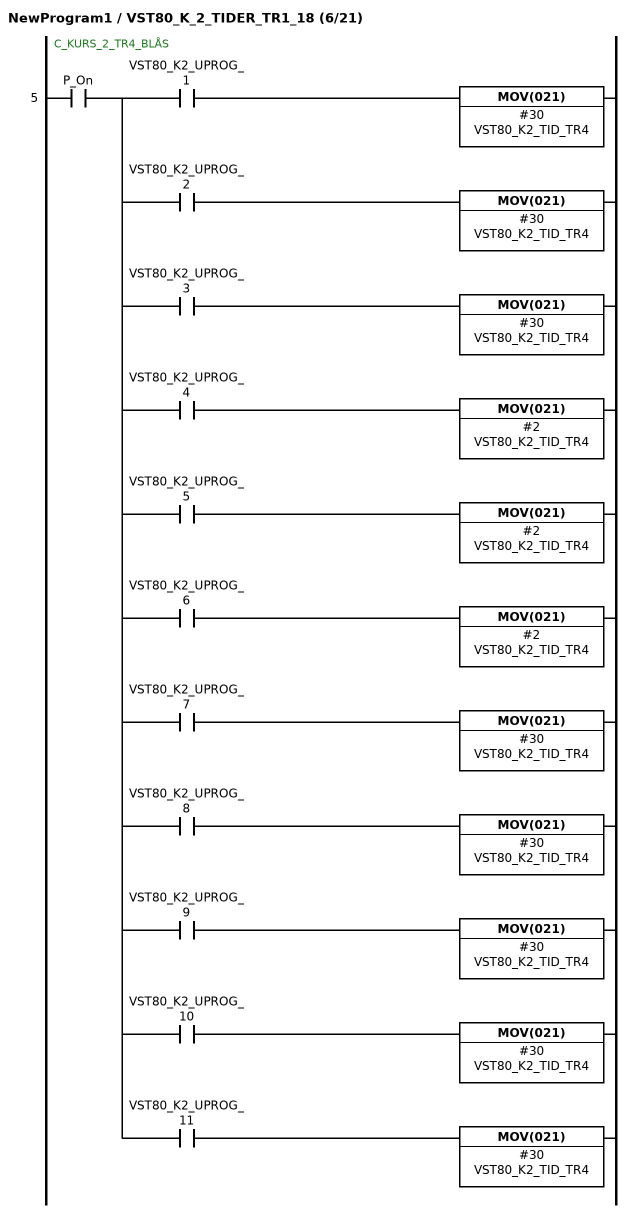
; [picture p168: NewProgram1 / VST80_K_2_TIDER_TR1_18, rungs 5-5]
; rung 5: C_KURS_2_TR4_BLÅS
LD P_On
OUT TR0
AND VST80_K2_UPROG_1
MOV(021) #30 VST80_K2_TID_TR4
LD TR0
AND VST80_K2_UPROG_2
MOV(021) #30 VST80_K2_TID_TR4
LD TR0
AND VST80_K2_UPROG_3
MOV(021) #30 VST80_K2_TID_TR4
LD TR0
AND VST80_K2_UPROG_4
MOV(021) #2 VST80_K2_TID_TR4
LD TR0
AND VST80_K2_UPROG_5
MOV(021) #2 VST80_K2_TID_TR4
LD TR0
AND VST80_K2_UPROG_6
MOV(021) #2 VST80_K2_TID_TR4
LD TR0
AND VST80_K2_UPROG_7
MOV(021) #30 VST80_K2_TID_TR4
LD TR0
AND VST80_K2_UPROG_8
MOV(021) #30 VST80_K2_TID_TR4
LD TR0
AND VST80_K2_UPROG_9
MOV(021) #30 VST80_K2_TID_TR4
LD TR0
AND VST80_K2_UPROG_10
MOV(021) #30 VST80_K2_TID_TR4
LD TR0
AND VST80_K2_UPROG_11
MOV(021) #30 VST80_K2_TID_TR4

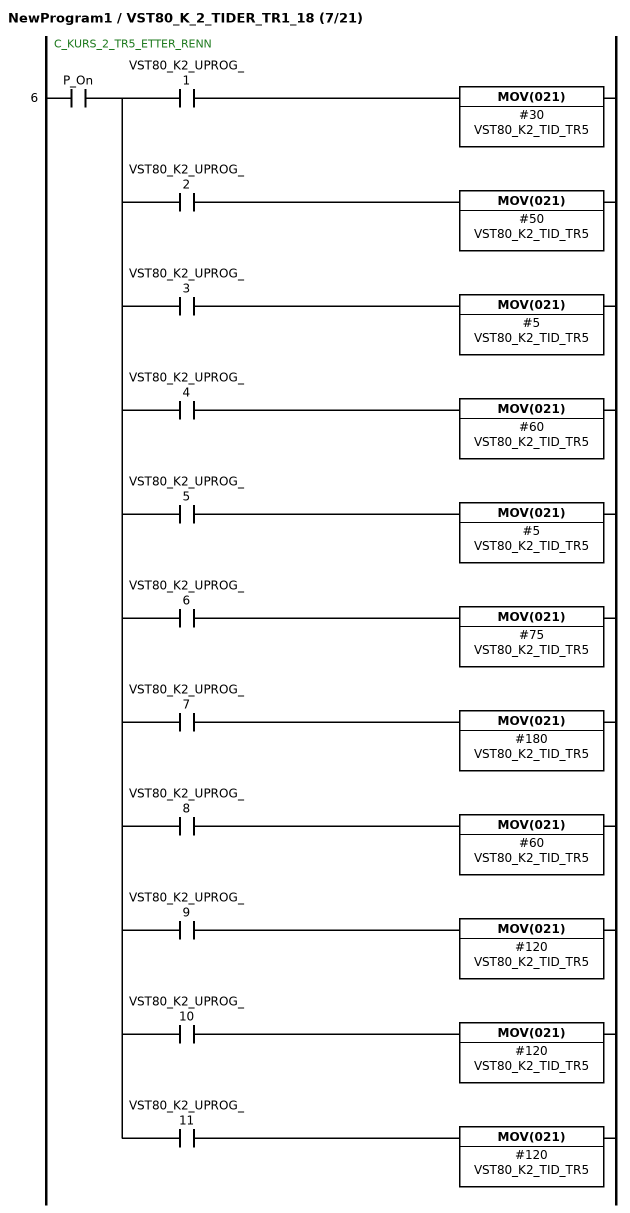
; rung 6: C_KURS_2_TR5_ETTER_RENN
LD P_On
OUT TR0
AND VST80_K2_UPROG_1
MOV(021) #30 VST80_K2_TID_TR5
LD TR0
AND VST80_K2_UPROG_2
MOV(021) #50 VST80_K2_TID_TR5
LD TR0
AND VST80_K2_UPROG_3
MOV(021) #5 VST80_K2_TID_TR5
LD TR0
AND VST80_K2_UPROG_4
MOV(021) #60 VST80_K2_TID_TR5
LD TR0
AND VST80_K2_UPROG_5
MOV(021) #5 VST80_K2_TID_TR5
LD TR0
AND VST80_K2_UPROG_6
MOV(021) #75 VST80_K2_TID_TR5
LD TR0
AND VST80_K2_UPROG_7
MOV(021) #180 VST80_K2_TID_TR5
LD TR0
AND VST80_K2_UPROG_8
MOV(021) #60 VST80_K2_TID_TR5
LD TR0
AND VST80_K2_UPROG_9
MOV(021) #120 VST80_K2_TID_TR5
LD TR0
AND VST80_K2_UPROG_10
MOV(021) #120 VST80_K2_TID_TR5
LD TR0
AND VST80_K2_UPROG_11
MOV(021) #120 VST80_K2_TID_TR5

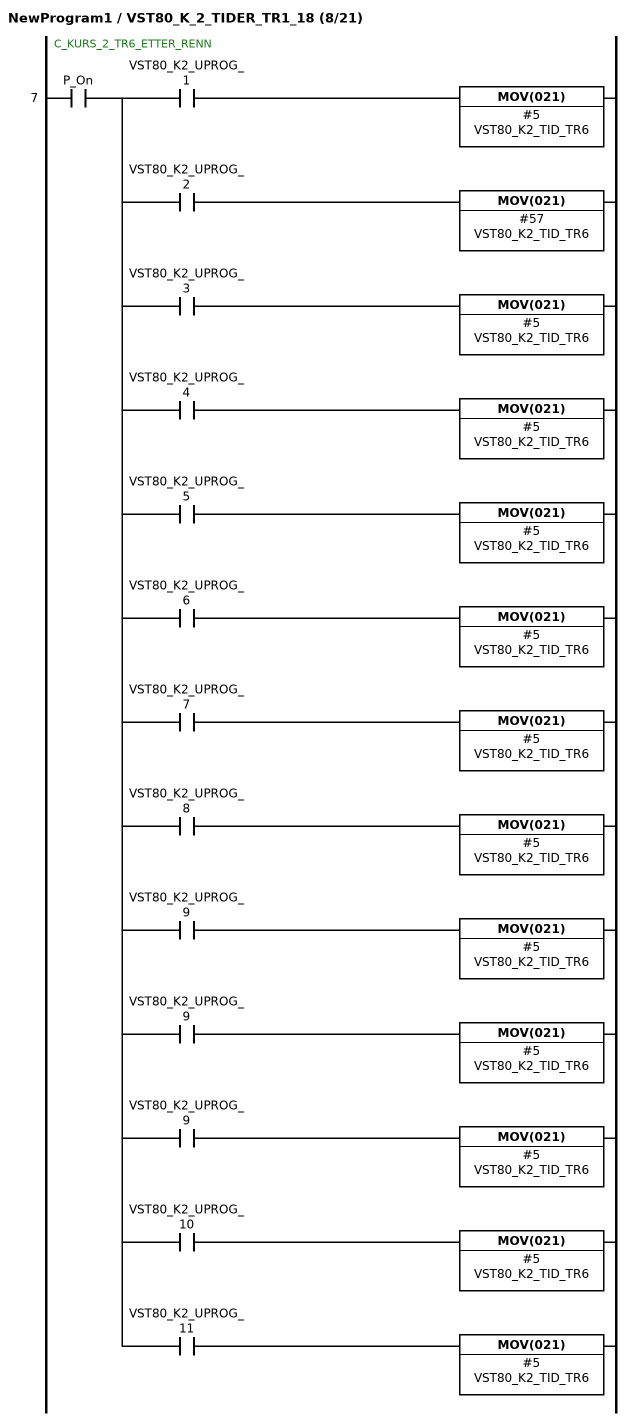
; rung 7: C_KURS_2_TR6_ETTER_RENN
LD P_On
OUT TR0
AND VST80_K2_UPROG_1
MOV(021) #5 VST80_K2_TID_TR6
LD TR0
AND VST80_K2_UPROG_2
MOV(021) #57 VST80_K2_TID_TR6
LD TR0
AND VST80_K2_UPROG_3
MOV(021) #5 VST80_K2_TID_TR6
LD TR0
AND VST80_K2_UPROG_4
MOV(021) #5 VST80_K2_TID_TR6
LD TR0
AND VST80_K2_UPROG_5
MOV(021) #5 VST80_K2_TID_TR6
LD TR0
AND VST80_K2_UPROG_6
MOV(021) #5 VST80_K2_TID_TR6
LD TR0
AND VST80_K2_UPROG_7
MOV(021) #5 VST80_K2_TID_TR6
LD TR0
AND VST80_K2_UPROG_8
MOV(021) #5 VST80_K2_TID_TR6
LD TR0
AND VST80_K2_UPROG_9
MOV(021) #5 VST80_K2_TID_TR6
LD TR0
AND VST80_K2_UPROG_9
MOV(021) #5 VST80_K2_TID_TR6
LD TR0
AND VST80_K2_UPROG_9
MOV(021) #5 VST80_K2_TID_TR6
LD TR0
AND VST80_K2_UPROG_10
MOV(021) #5 VST80_K2_TID_TR6
LD TR0
AND VST80_K2_UPROG_11
MOV(021) #5 VST80_K2_TID_TR6

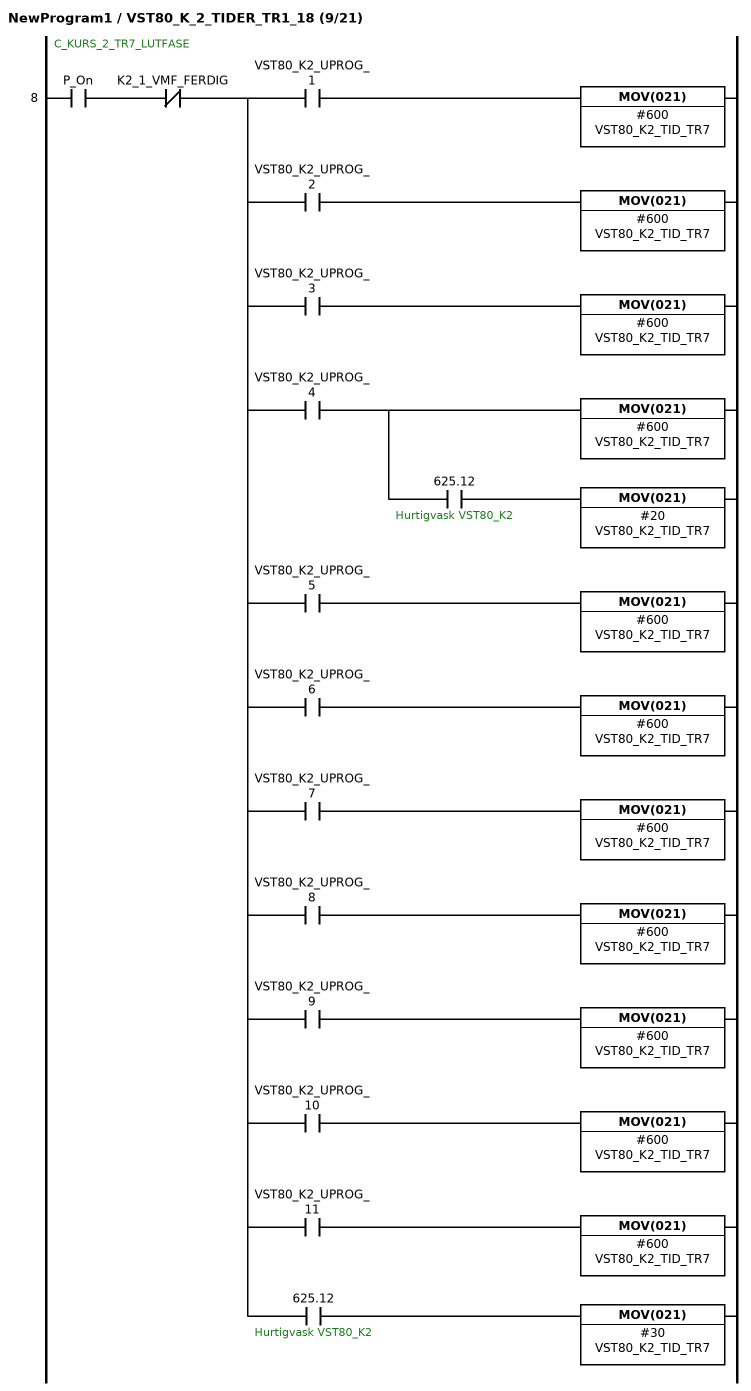
; rung 8: C_KURS_2_TR7_LUTFASE
LD P_On
ANDNOT K2_1_VMF_FERDIG
OUT TR0
AND VST80_K2_UPROG_1
MOV(021) #600 VST80_K2_TID_TR7
LD TR0
AND VST80_K2_UPROG_2
MOV(021) #600 VST80_K2_TID_TR7
LD TR0
AND VST80_K2_UPROG_3
MOV(021) #600 VST80_K2_TID_TR7
LD TR0
AND VST80_K2_UPROG_4
MOV(021) #600 VST80_K2_TID_TR7
AND 625.12  ; Hurtigvask VST80_K2
MOV(021) #20 VST80_K2_TID_TR7
LD TR0
AND VST80_K2_UPROG_5
MOV(021) #600 VST80_K2_TID_TR7
LD TR0
AND VST80_K2_UPROG_6
MOV(021) #600 VST80_K2_TID_TR7
LD TR0
AND VST80_K2_UPROG_7
MOV(021) #600 VST80_K2_TID_TR7
LD TR0
AND VST80_K2_UPROG_8
MOV(021) #600 VST80_K2_TID_TR7
LD TR0
AND VST80_K2_UPROG_9
MOV(021) #600 VST80_K2_TID_TR7
LD TR0
AND VST80_K2_UPROG_10
MOV(021) #600 VST80_K2_TID_TR7
LD TR0
AND VST80_K2_UPROG_11
MOV(021) #600 VST80_K2_TID_TR7
LD TR0
AND 625.12  ; Hurtigvask VST80_K2
MOV(021) #30 VST80_K2_TID_TR7

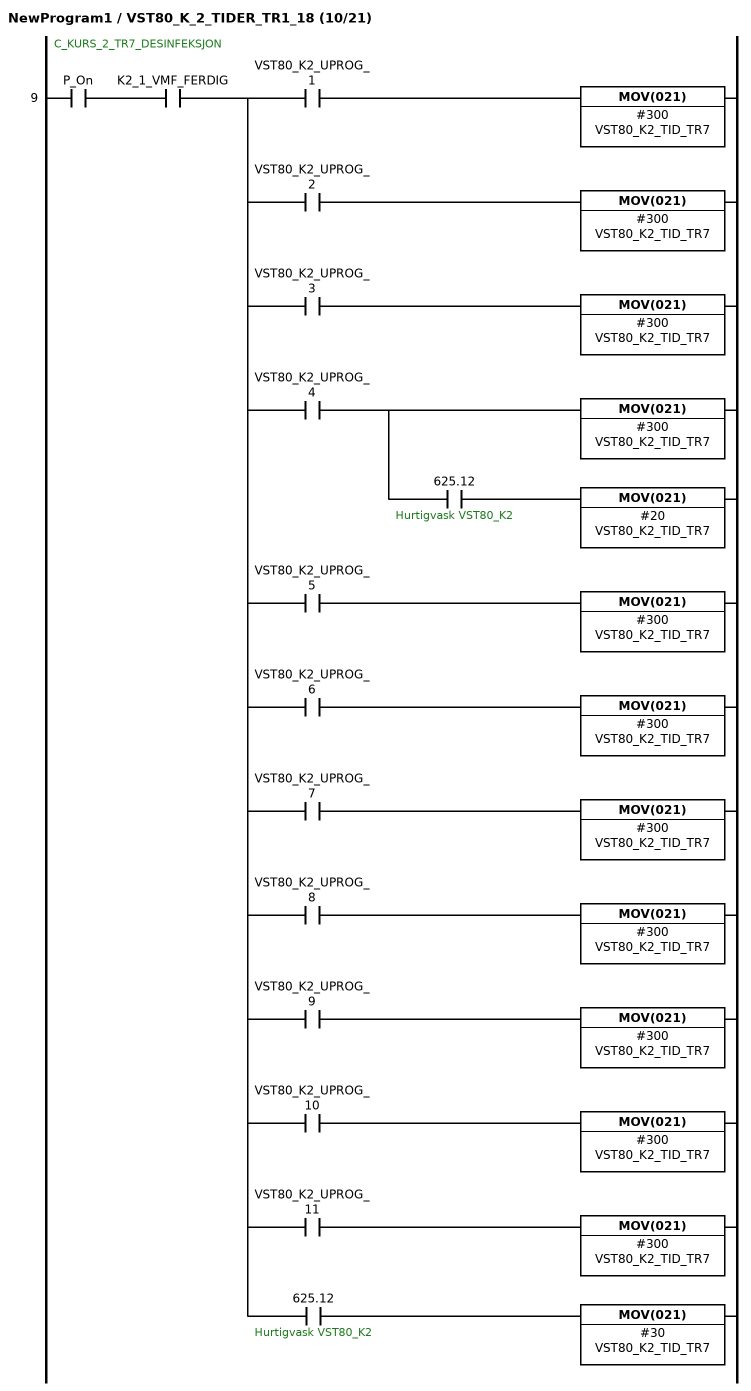
; rung 9: C_KURS_2_TR7_DESINFEKSJON
LD P_On
AND K2_1_VMF_FERDIG
OUT TR0
AND VST80_K2_UPROG_1
MOV(021) #300 VST80_K2_TID_TR7
LD TR0
AND VST80_K2_UPROG_2
MOV(021) #300 VST80_K2_TID_TR7
LD TR0
AND VST80_K2_UPROG_3
MOV(021) #300 VST80_K2_TID_TR7
LD TR0
AND VST80_K2_UPROG_4
MOV(021) #300 VST80_K2_TID_TR7
AND 625.12  ; Hurtigvask VST80_K2
MOV(021) #20 VST80_K2_TID_TR7
LD TR0
AND VST80_K2_UPROG_5
MOV(021) #300 VST80_K2_TID_TR7
LD TR0
AND VST80_K2_UPROG_6
MOV(021) #300 VST80_K2_TID_TR7
LD TR0
AND VST80_K2_UPROG_7
MOV(021) #300 VST80_K2_TID_TR7
LD TR0
AND VST80_K2_UPROG_8
MOV(021) #300 VST80_K2_TID_TR7
LD TR0
AND VST80_K2_UPROG_9
MOV(021) #300 VST80_K2_TID_TR7
LD TR0
AND VST80_K2_UPROG_10
MOV(021) #300 VST80_K2_TID_TR7
LD TR0
AND VST80_K2_UPROG_11
MOV(021) #300 VST80_K2_TID_TR7
LD TR0
AND 625.12  ; Hurtigvask VST80_K2
MOV(021) #30 VST80_K2_TID_TR7

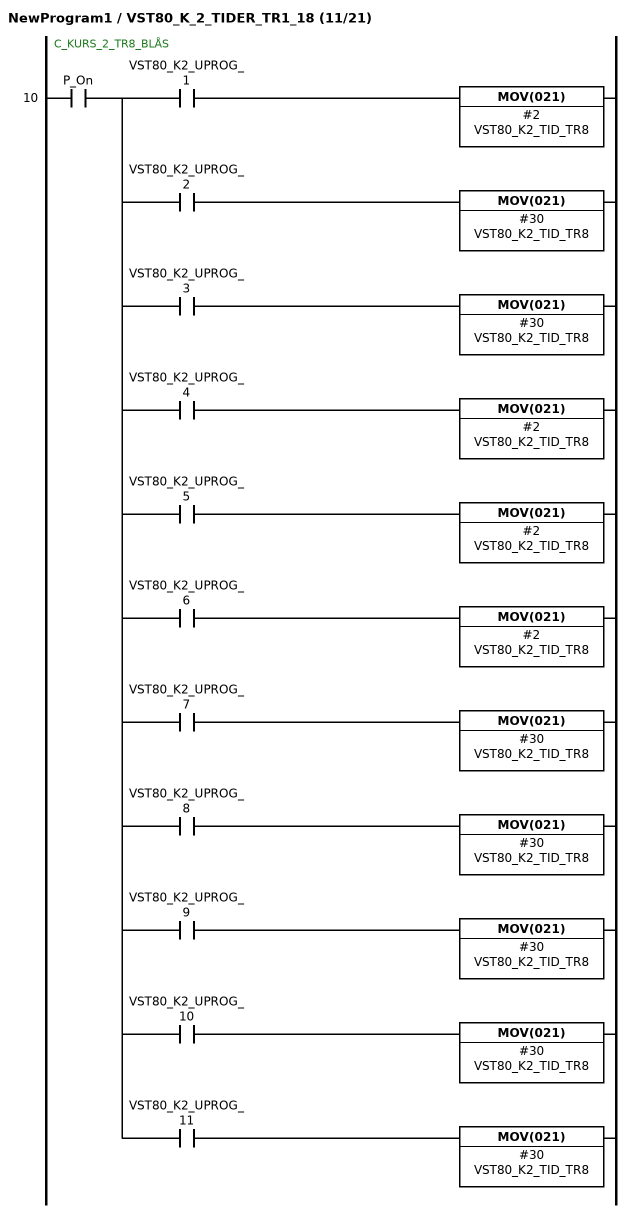
; rung 10: C_KURS_2_TR8_BLÅS
LD P_On
OUT TR0
AND VST80_K2_UPROG_1
MOV(021) #2 VST80_K2_TID_TR8
LD TR0
AND VST80_K2_UPROG_2
MOV(021) #30 VST80_K2_TID_TR8
LD TR0
AND VST80_K2_UPROG_3
MOV(021) #30 VST80_K2_TID_TR8
LD TR0
AND VST80_K2_UPROG_4
MOV(021) #2 VST80_K2_TID_TR8
LD TR0
AND VST80_K2_UPROG_5
MOV(021) #2 VST80_K2_TID_TR8
LD TR0
AND VST80_K2_UPROG_6
MOV(021) #2 VST80_K2_TID_TR8
LD TR0
AND VST80_K2_UPROG_7
MOV(021) #30 VST80_K2_TID_TR8
LD TR0
AND VST80_K2_UPROG_8
MOV(021) #30 VST80_K2_TID_TR8
LD TR0
AND VST80_K2_UPROG_9
MOV(021) #30 VST80_K2_TID_TR8
LD TR0
AND VST80_K2_UPROG_10
MOV(021) #30 VST80_K2_TID_TR8
LD TR0
AND VST80_K2_UPROG_11
MOV(021) #30 VST80_K2_TID_TR8

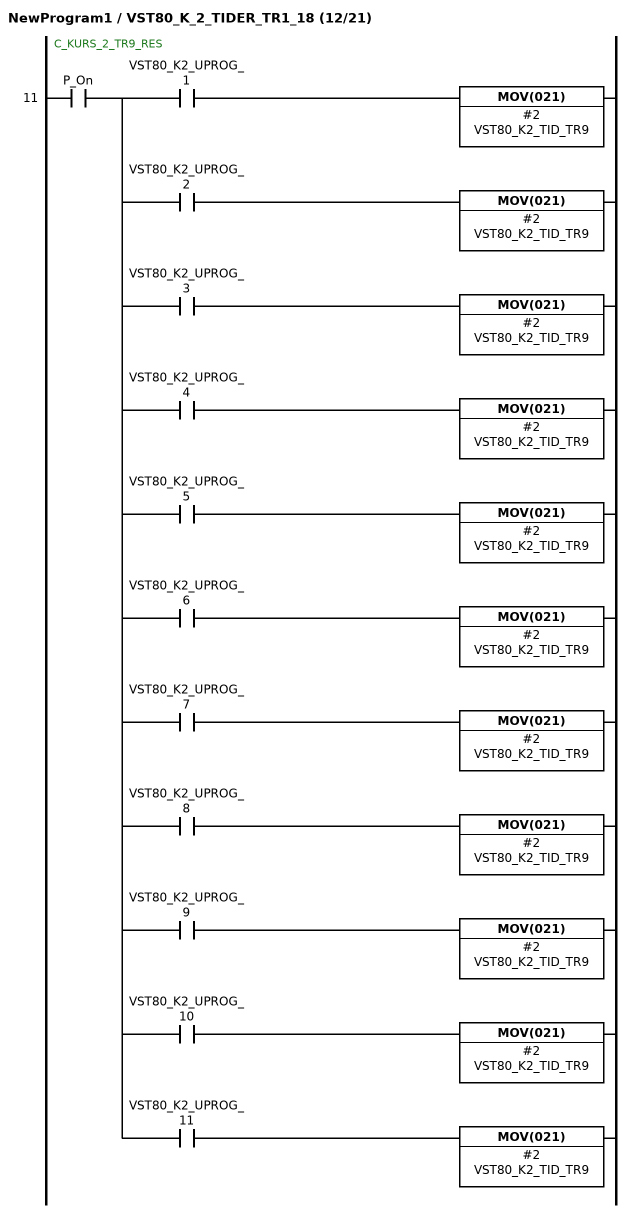
; rung 11: C_KURS_2_TR9_RES
LD P_On
OUT TR0
AND VST80_K2_UPROG_1
MOV(021) #2 VST80_K2_TID_TR9
LD TR0
AND VST80_K2_UPROG_2
MOV(021) #2 VST80_K2_TID_TR9
LD TR0
AND VST80_K2_UPROG_3
MOV(021) #2 VST80_K2_TID_TR9
LD TR0
AND VST80_K2_UPROG_4
MOV(021) #2 VST80_K2_TID_TR9
LD TR0
AND VST80_K2_UPROG_5
MOV(021) #2 VST80_K2_TID_TR9
LD TR0
AND VST80_K2_UPROG_6
MOV(021) #2 VST80_K2_TID_TR9
LD TR0
AND VST80_K2_UPROG_7
MOV(021) #2 VST80_K2_TID_TR9
LD TR0
AND VST80_K2_UPROG_8
MOV(021) #2 VST80_K2_TID_TR9
LD TR0
AND VST80_K2_UPROG_9
MOV(021) #2 VST80_K2_TID_TR9
LD TR0
AND VST80_K2_UPROG_10
MOV(021) #2 VST80_K2_TID_TR9
LD TR0
AND VST80_K2_UPROG_11
MOV(021) #2 VST80_K2_TID_TR9

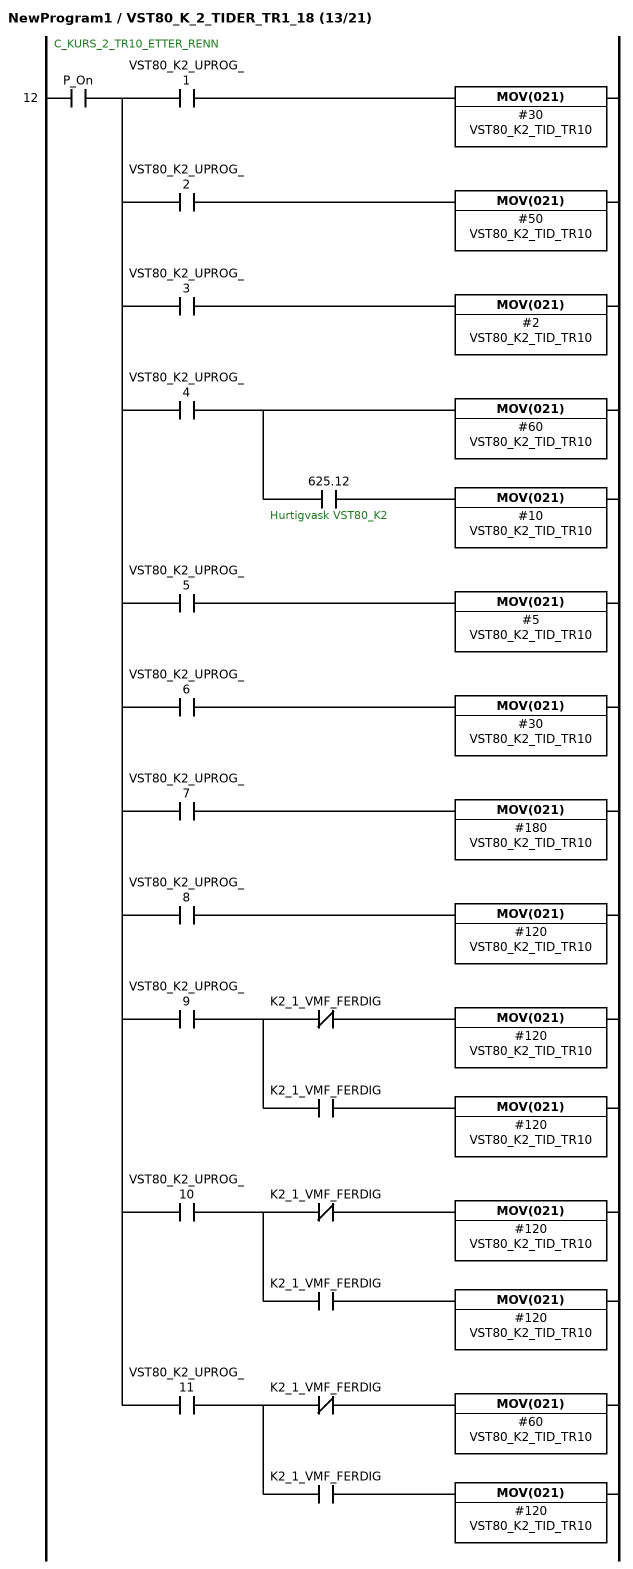
; rung 12: C_KURS_2_TR10_ETTER_RENN
LD P_On
OUT TR0
AND VST80_K2_UPROG_1
MOV(021) #30 VST80_K2_TID_TR10
LD TR0
AND VST80_K2_UPROG_2
MOV(021) #50 VST80_K2_TID_TR10
LD TR0
AND VST80_K2_UPROG_3
MOV(021) #2 VST80_K2_TID_TR10
LD TR0
AND VST80_K2_UPROG_4
MOV(021) #60 VST80_K2_TID_TR10
AND 625.12  ; Hurtigvask VST80_K2
MOV(021) #10 VST80_K2_TID_TR10
LD TR0
AND VST80_K2_UPROG_5
MOV(021) #5 VST80_K2_TID_TR10
LD TR0
AND VST80_K2_UPROG_6
MOV(021) #30 VST80_K2_TID_TR10
LD TR0
AND VST80_K2_UPROG_7
MOV(021) #180 VST80_K2_TID_TR10
LD TR0
AND VST80_K2_UPROG_8
MOV(021) #120 VST80_K2_TID_TR10
LD TR0
AND VST80_K2_UPROG_9
OUT TR1
ANDNOT K2_1_VMF_FERDIG
MOV(021) #120 VST80_K2_TID_TR10
LD TR1
AND K2_1_VMF_FERDIG
MOV(021) #120 VST80_K2_TID_TR10
LD TR0
AND VST80_K2_UPROG_10
OUT TR1
ANDNOT K2_1_VMF_FERDIG
MOV(021) #120 VST80_K2_TID_TR10
LD TR1
AND K2_1_VMF_FERDIG
MOV(021) #120 VST80_K2_TID_TR10
LD TR0
AND VST80_K2_UPROG_11
OUT TR0
ANDNOT K2_1_VMF_FERDIG
MOV(021) #60 VST80_K2_TID_TR10
LD TR0
AND K2_1_VMF_FERDIG
MOV(021) #120 VST80_K2_TID_TR10

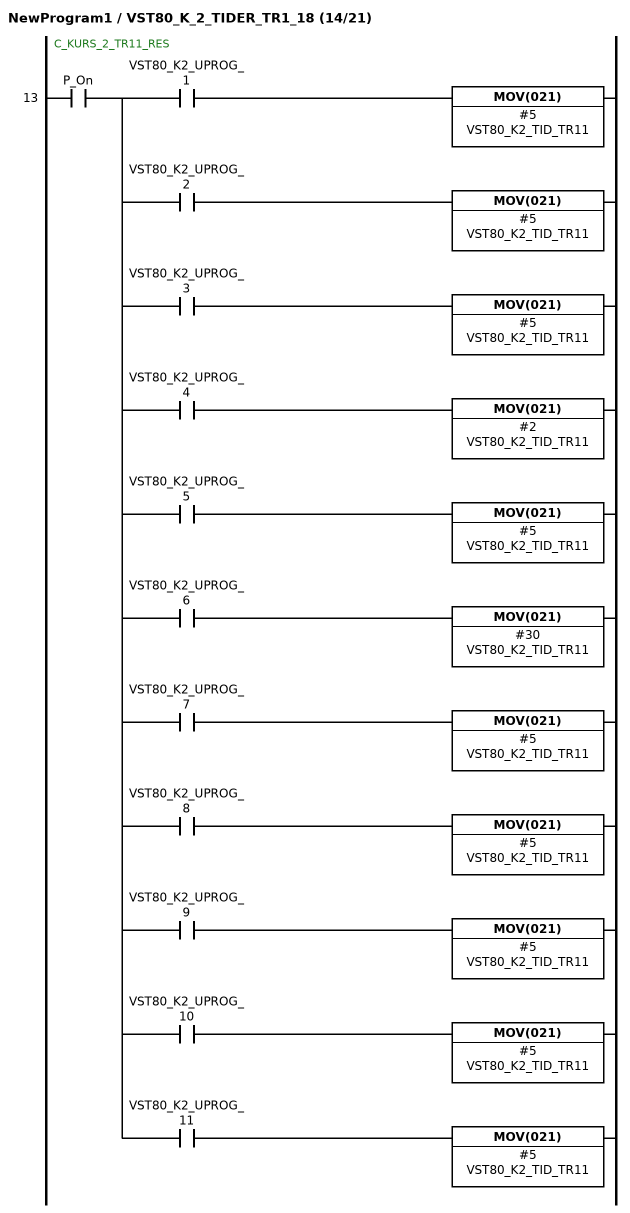
; rung 13: C_KURS_2_TR11_RES
LD P_On
OUT TR0
AND VST80_K2_UPROG_1
MOV(021) #5 VST80_K2_TID_TR11
LD TR0
AND VST80_K2_UPROG_2
MOV(021) #5 VST80_K2_TID_TR11
LD TR0
AND VST80_K2_UPROG_3
MOV(021) #5 VST80_K2_TID_TR11
LD TR0
AND VST80_K2_UPROG_4
MOV(021) #2 VST80_K2_TID_TR11
LD TR0
AND VST80_K2_UPROG_5
MOV(021) #5 VST80_K2_TID_TR11
LD TR0
AND VST80_K2_UPROG_6
MOV(021) #30 VST80_K2_TID_TR11
LD TR0
AND VST80_K2_UPROG_7
MOV(021) #5 VST80_K2_TID_TR11
LD TR0
AND VST80_K2_UPROG_8
MOV(021) #5 VST80_K2_TID_TR11
LD TR0
AND VST80_K2_UPROG_9
MOV(021) #5 VST80_K2_TID_TR11
LD TR0
AND VST80_K2_UPROG_10
MOV(021) #5 VST80_K2_TID_TR11
LD TR0
AND VST80_K2_UPROG_11
MOV(021) #5 VST80_K2_TID_TR11

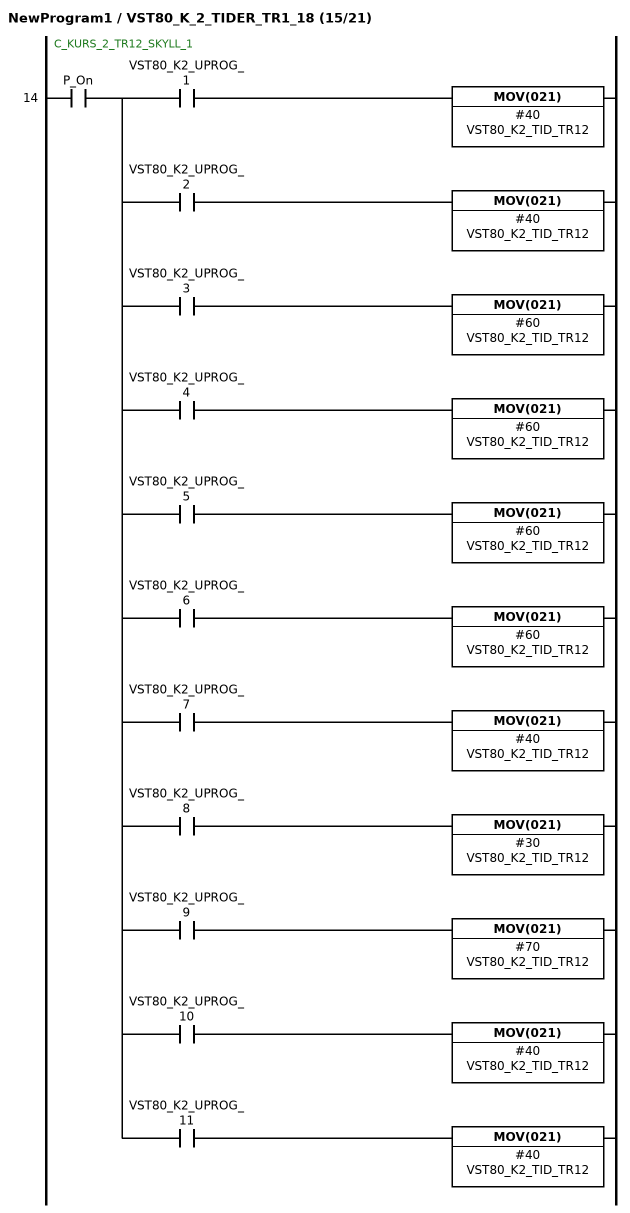
; rung 14: C_KURS_2_TR12_SKYLL_1
LD P_On
OUT TR0
AND VST80_K2_UPROG_1
MOV(021) #40 VST80_K2_TID_TR12
LD TR0
AND VST80_K2_UPROG_2
MOV(021) #40 VST80_K2_TID_TR12
LD TR0
AND VST80_K2_UPROG_3
MOV(021) #60 VST80_K2_TID_TR12
LD TR0
AND VST80_K2_UPROG_4
MOV(021) #60 VST80_K2_TID_TR12
LD TR0
AND VST80_K2_UPROG_5
MOV(021) #60 VST80_K2_TID_TR12
LD TR0
AND VST80_K2_UPROG_6
MOV(021) #60 VST80_K2_TID_TR12
LD TR0
AND VST80_K2_UPROG_7
MOV(021) #40 VST80_K2_TID_TR12
LD TR0
AND VST80_K2_UPROG_8
MOV(021) #30 VST80_K2_TID_TR12
LD TR0
AND VST80_K2_UPROG_9
MOV(021) #70 VST80_K2_TID_TR12
LD TR0
AND VST80_K2_UPROG_10
MOV(021) #40 VST80_K2_TID_TR12
LD TR0
AND VST80_K2_UPROG_11
MOV(021) #40 VST80_K2_TID_TR12

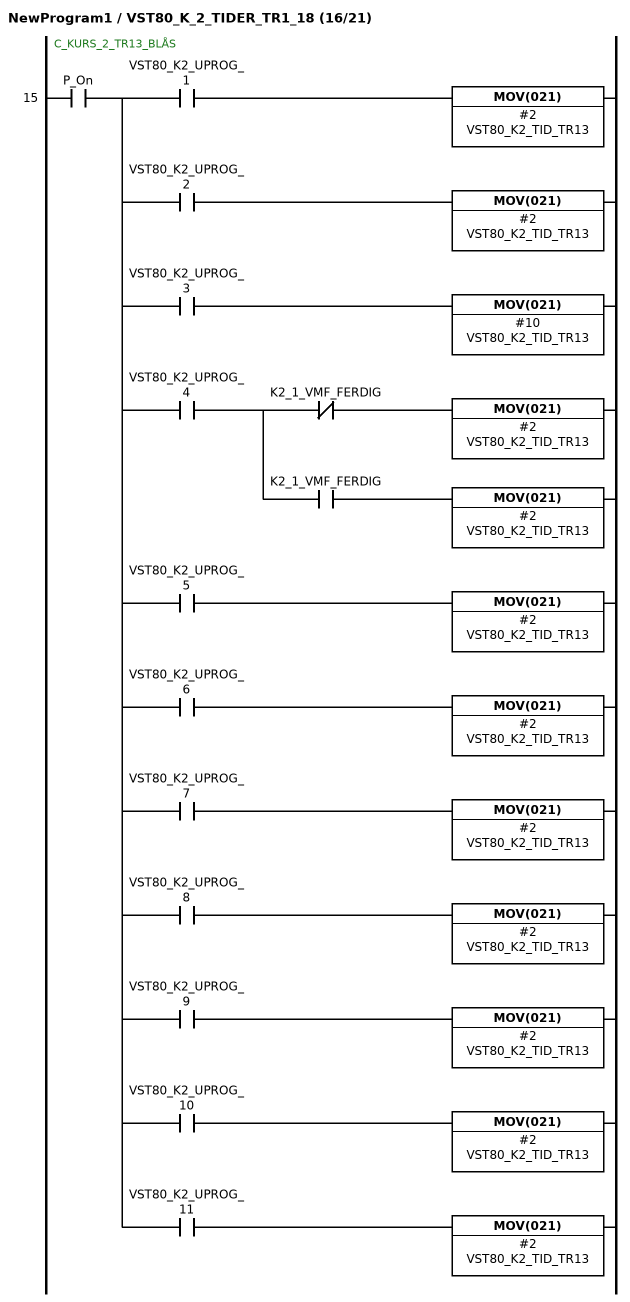
; rung 15: C_KURS_2_TR13_BLÅS
LD P_On
OUT TR0
AND VST80_K2_UPROG_1
MOV(021) #2 VST80_K2_TID_TR13
LD TR0
AND VST80_K2_UPROG_2
MOV(021) #2 VST80_K2_TID_TR13
LD TR0
AND VST80_K2_UPROG_3
MOV(021) #10 VST80_K2_TID_TR13
LD TR0
AND VST80_K2_UPROG_4
OUT TR1
ANDNOT K2_1_VMF_FERDIG
MOV(021) #2 VST80_K2_TID_TR13
LD TR1
AND K2_1_VMF_FERDIG
MOV(021) #2 VST80_K2_TID_TR13
LD TR0
AND VST80_K2_UPROG_5
MOV(021) #2 VST80_K2_TID_TR13
LD TR0
AND VST80_K2_UPROG_6
MOV(021) #2 VST80_K2_TID_TR13
LD TR0
AND VST80_K2_UPROG_7
MOV(021) #2 VST80_K2_TID_TR13
LD TR0
AND VST80_K2_UPROG_8
MOV(021) #2 VST80_K2_TID_TR13
LD TR0
AND VST80_K2_UPROG_9
MOV(021) #2 VST80_K2_TID_TR13
LD TR0
AND VST80_K2_UPROG_10
MOV(021) #2 VST80_K2_TID_TR13
LD TR0
AND VST80_K2_UPROG_11
MOV(021) #2 VST80_K2_TID_TR13

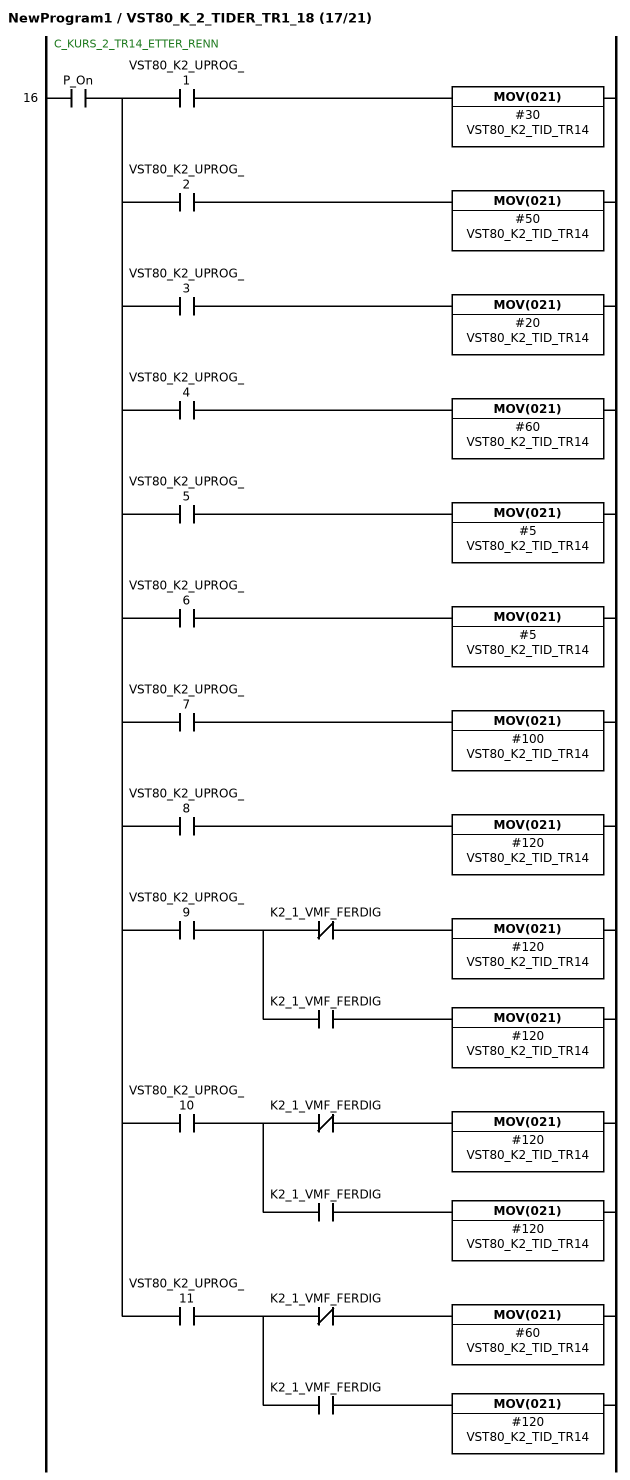
; rung 16: C_KURS_2_TR14_ETTER_RENN
LD P_On
OUT TR0
AND VST80_K2_UPROG_1
MOV(021) #30 VST80_K2_TID_TR14
LD TR0
AND VST80_K2_UPROG_2
MOV(021) #50 VST80_K2_TID_TR14
LD TR0
AND VST80_K2_UPROG_3
MOV(021) #20 VST80_K2_TID_TR14
LD TR0
AND VST80_K2_UPROG_4
MOV(021) #60 VST80_K2_TID_TR14
LD TR0
AND VST80_K2_UPROG_5
MOV(021) #5 VST80_K2_TID_TR14
LD TR0
AND VST80_K2_UPROG_6
MOV(021) #5 VST80_K2_TID_TR14
LD TR0
AND VST80_K2_UPROG_7
MOV(021) #100 VST80_K2_TID_TR14
LD TR0
AND VST80_K2_UPROG_8
MOV(021) #120 VST80_K2_TID_TR14
LD TR0
AND VST80_K2_UPROG_9
OUT TR1
ANDNOT K2_1_VMF_FERDIG
MOV(021) #120 VST80_K2_TID_TR14
LD TR1
AND K2_1_VMF_FERDIG
MOV(021) #120 VST80_K2_TID_TR14
LD TR0
AND VST80_K2_UPROG_10
OUT TR1
ANDNOT K2_1_VMF_FERDIG
MOV(021) #120 VST80_K2_TID_TR14
LD TR1
AND K2_1_VMF_FERDIG
MOV(021) #120 VST80_K2_TID_TR14
LD TR0
AND VST80_K2_UPROG_11
OUT TR0
ANDNOT K2_1_VMF_FERDIG
MOV(021) #60 VST80_K2_TID_TR14
LD TR0
AND K2_1_VMF_FERDIG
MOV(021) #120 VST80_K2_TID_TR14

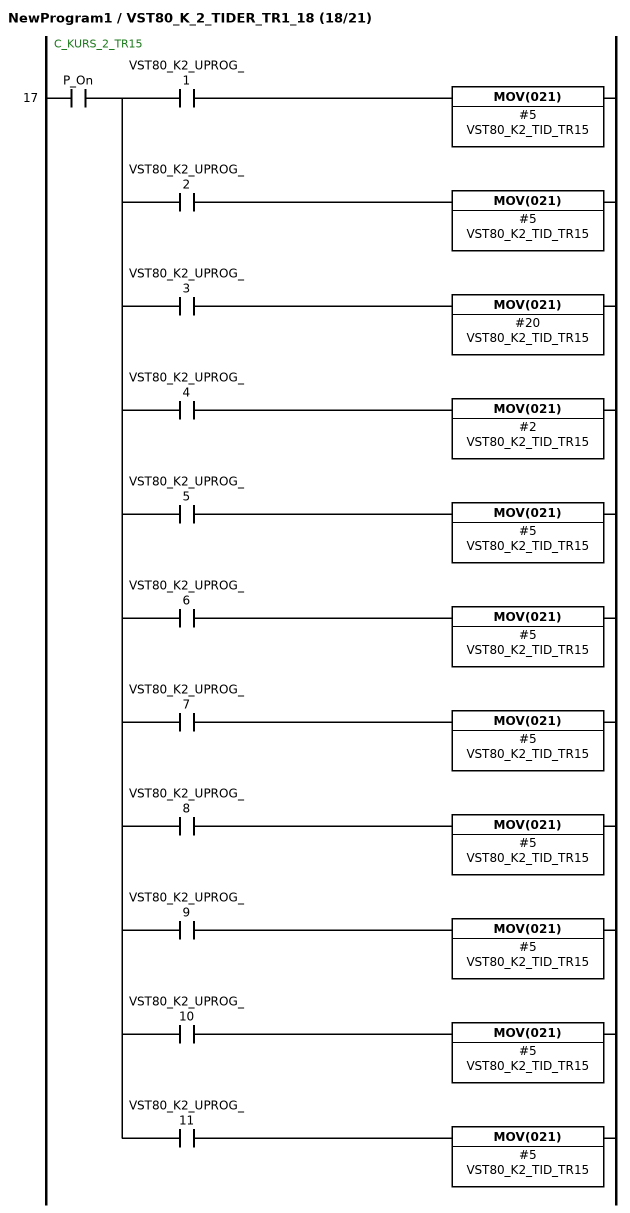
; rung 17: C_KURS_2_TR15
LD P_On
OUT TR0
AND VST80_K2_UPROG_1
MOV(021) #5 VST80_K2_TID_TR15
LD TR0
AND VST80_K2_UPROG_2
MOV(021) #5 VST80_K2_TID_TR15
LD TR0
AND VST80_K2_UPROG_3
MOV(021) #20 VST80_K2_TID_TR15
LD TR0
AND VST80_K2_UPROG_4
MOV(021) #2 VST80_K2_TID_TR15
LD TR0
AND VST80_K2_UPROG_5
MOV(021) #5 VST80_K2_TID_TR15
LD TR0
AND VST80_K2_UPROG_6
MOV(021) #5 VST80_K2_TID_TR15
LD TR0
AND VST80_K2_UPROG_7
MOV(021) #5 VST80_K2_TID_TR15
LD TR0
AND VST80_K2_UPROG_8
MOV(021) #5 VST80_K2_TID_TR15
LD TR0
AND VST80_K2_UPROG_9
MOV(021) #5 VST80_K2_TID_TR15
LD TR0
AND VST80_K2_UPROG_10
MOV(021) #5 VST80_K2_TID_TR15
LD TR0
AND VST80_K2_UPROG_11
MOV(021) #5 VST80_K2_TID_TR15

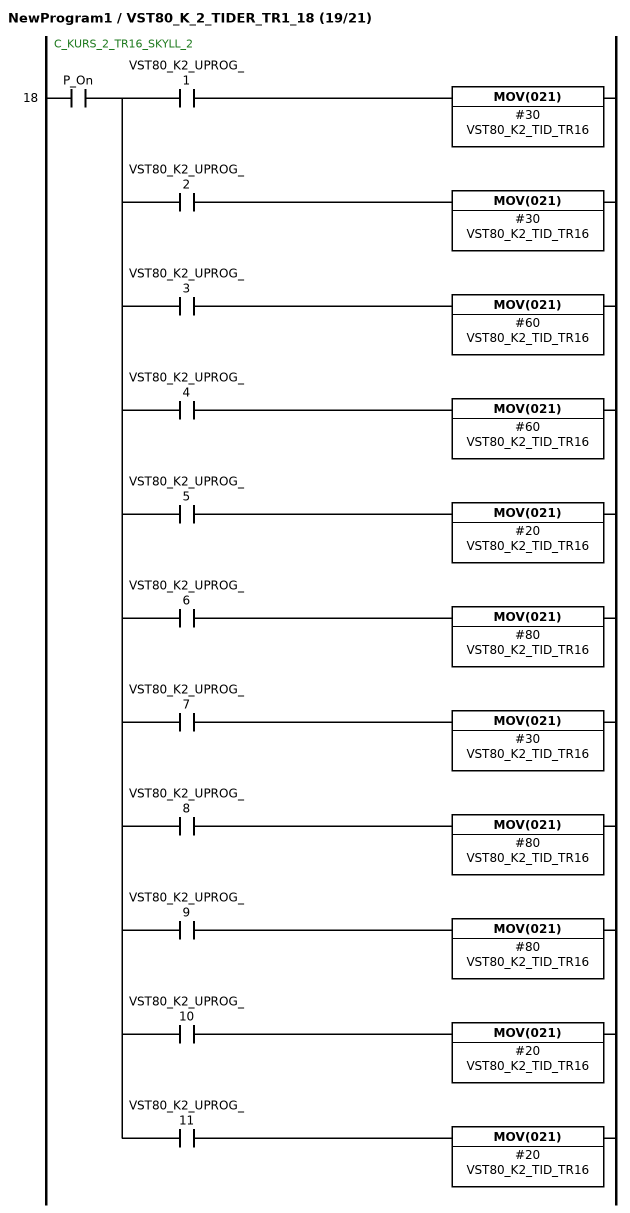
; rung 18: C_KURS_2_TR16_SKYLL_2
LD P_On
OUT TR0
AND VST80_K2_UPROG_1
MOV(021) #30 VST80_K2_TID_TR16
LD TR0
AND VST80_K2_UPROG_2
MOV(021) #30 VST80_K2_TID_TR16
LD TR0
AND VST80_K2_UPROG_3
MOV(021) #60 VST80_K2_TID_TR16
LD TR0
AND VST80_K2_UPROG_4
MOV(021) #60 VST80_K2_TID_TR16
LD TR0
AND VST80_K2_UPROG_5
MOV(021) #20 VST80_K2_TID_TR16
LD TR0
AND VST80_K2_UPROG_6
MOV(021) #80 VST80_K2_TID_TR16
LD TR0
AND VST80_K2_UPROG_7
MOV(021) #30 VST80_K2_TID_TR16
LD TR0
AND VST80_K2_UPROG_8
MOV(021) #80 VST80_K2_TID_TR16
LD TR0
AND VST80_K2_UPROG_9
MOV(021) #80 VST80_K2_TID_TR16
LD TR0
AND VST80_K2_UPROG_10
MOV(021) #20 VST80_K2_TID_TR16
LD TR0
AND VST80_K2_UPROG_11
MOV(021) #20 VST80_K2_TID_TR16

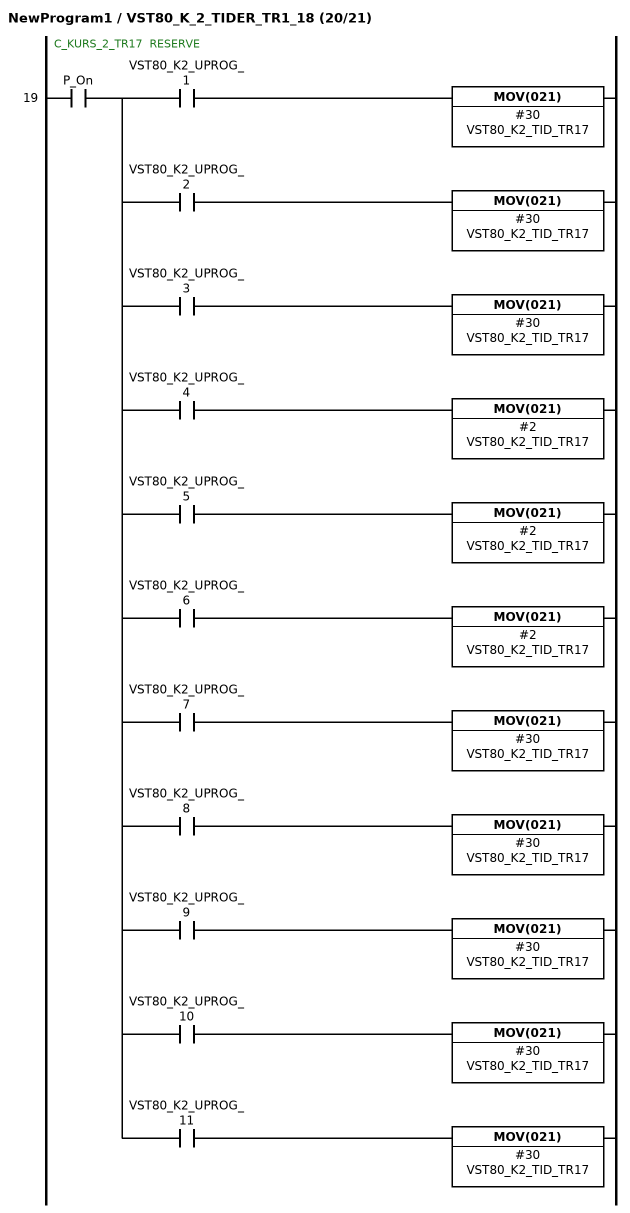
; rung 19: C_KURS_2_TR17  RESERVE
LD P_On
OUT TR0
AND VST80_K2_UPROG_1
MOV(021) #30 VST80_K2_TID_TR17
LD TR0
AND VST80_K2_UPROG_2
MOV(021) #30 VST80_K2_TID_TR17
LD TR0
AND VST80_K2_UPROG_3
MOV(021) #30 VST80_K2_TID_TR17
LD TR0
AND VST80_K2_UPROG_4
MOV(021) #2 VST80_K2_TID_TR17
LD TR0
AND VST80_K2_UPROG_5
MOV(021) #2 VST80_K2_TID_TR17
LD TR0
AND VST80_K2_UPROG_6
MOV(021) #2 VST80_K2_TID_TR17
LD TR0
AND VST80_K2_UPROG_7
MOV(021) #30 VST80_K2_TID_TR17
LD TR0
AND VST80_K2_UPROG_8
MOV(021) #30 VST80_K2_TID_TR17
LD TR0
AND VST80_K2_UPROG_9
MOV(021) #30 VST80_K2_TID_TR17
LD TR0
AND VST80_K2_UPROG_10
MOV(021) #30 VST80_K2_TID_TR17
LD TR0
AND VST80_K2_UPROG_11
MOV(021) #30 VST80_K2_TID_TR17

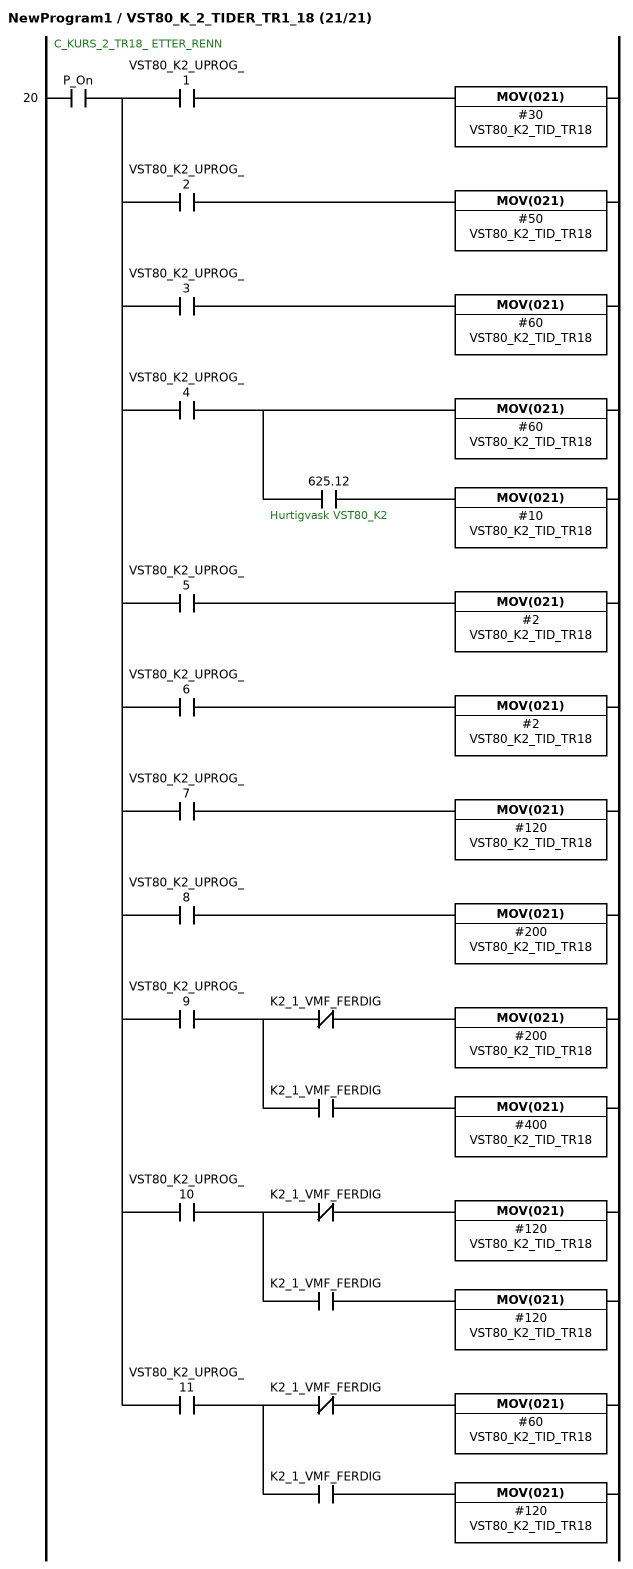
; rung 20: C_KURS_2_TR18_ ETTER_RENN
LD P_On
OUT TR0
AND VST80_K2_UPROG_1
MOV(021) #30 VST80_K2_TID_TR18
LD TR0
AND VST80_K2_UPROG_2
MOV(021) #50 VST80_K2_TID_TR18
LD TR0
AND VST80_K2_UPROG_3
MOV(021) #60 VST80_K2_TID_TR18
LD TR0
AND VST80_K2_UPROG_4
MOV(021) #60 VST80_K2_TID_TR18
AND 625.12  ; Hurtigvask VST80_K2
MOV(021) #10 VST80_K2_TID_TR18
LD TR0
AND VST80_K2_UPROG_5
MOV(021) #2 VST80_K2_TID_TR18
LD TR0
AND VST80_K2_UPROG_6
MOV(021) #2 VST80_K2_TID_TR18
LD TR0
AND VST80_K2_UPROG_7
MOV(021) #120 VST80_K2_TID_TR18
LD TR0
AND VST80_K2_UPROG_8
MOV(021) #200 VST80_K2_TID_TR18
LD TR0
AND VST80_K2_UPROG_9
OUT TR1
ANDNOT K2_1_VMF_FERDIG
MOV(021) #200 VST80_K2_TID_TR18
LD TR1
AND K2_1_VMF_FERDIG
MOV(021) #400 VST80_K2_TID_TR18
LD TR0
AND VST80_K2_UPROG_10
OUT TR1
ANDNOT K2_1_VMF_FERDIG
MOV(021) #120 VST80_K2_TID_TR18
LD TR1
AND K2_1_VMF_FERDIG
MOV(021) #120 VST80_K2_TID_TR18
LD TR0
AND VST80_K2_UPROG_11
OUT TR0
ANDNOT K2_1_VMF_FERDIG
MOV(021) #60 VST80_K2_TID_TR18
LD TR0
AND K2_1_VMF_FERDIG
MOV(021) #120 VST80_K2_TID_TR18
; rung 21: Ingen_kommentar_funnet

### Section VST80_K_2_TIDER_TR19_30

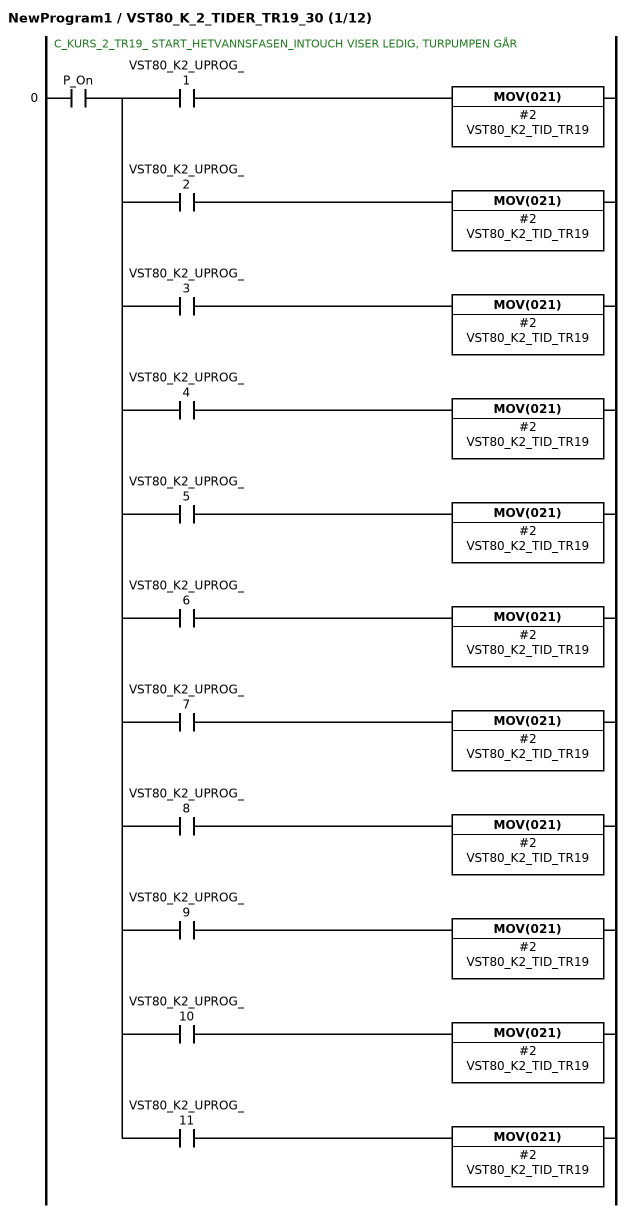
; rung 0: C_KURS_2_TR19_ START_HETVANNSFASEN_INTOUCH VISER LEDIG, TURPUMPEN GÅR
LD P_On
OUT TR0
AND VST80_K2_UPROG_1
MOV(021) #2 VST80_K2_TID_TR19
LD TR0
AND VST80_K2_UPROG_2
MOV(021) #2 VST80_K2_TID_TR19
LD TR0
AND VST80_K2_UPROG_3
MOV(021) #2 VST80_K2_TID_TR19
LD TR0
AND VST80_K2_UPROG_4
MOV(021) #2 VST80_K2_TID_TR19
LD TR0
AND VST80_K2_UPROG_5
MOV(021) #2 VST80_K2_TID_TR19
LD TR0
AND VST80_K2_UPROG_6
MOV(021) #2 VST80_K2_TID_TR19
LD TR0
AND VST80_K2_UPROG_7
MOV(021) #2 VST80_K2_TID_TR19
LD TR0
AND VST80_K2_UPROG_8
MOV(021) #2 VST80_K2_TID_TR19
LD TR0
AND VST80_K2_UPROG_9
MOV(021) #2 VST80_K2_TID_TR19
LD TR0
AND VST80_K2_UPROG_10
MOV(021) #2 VST80_K2_TID_TR19
LD TR0
AND VST80_K2_UPROG_11
MOV(021) #2 VST80_K2_TID_TR19

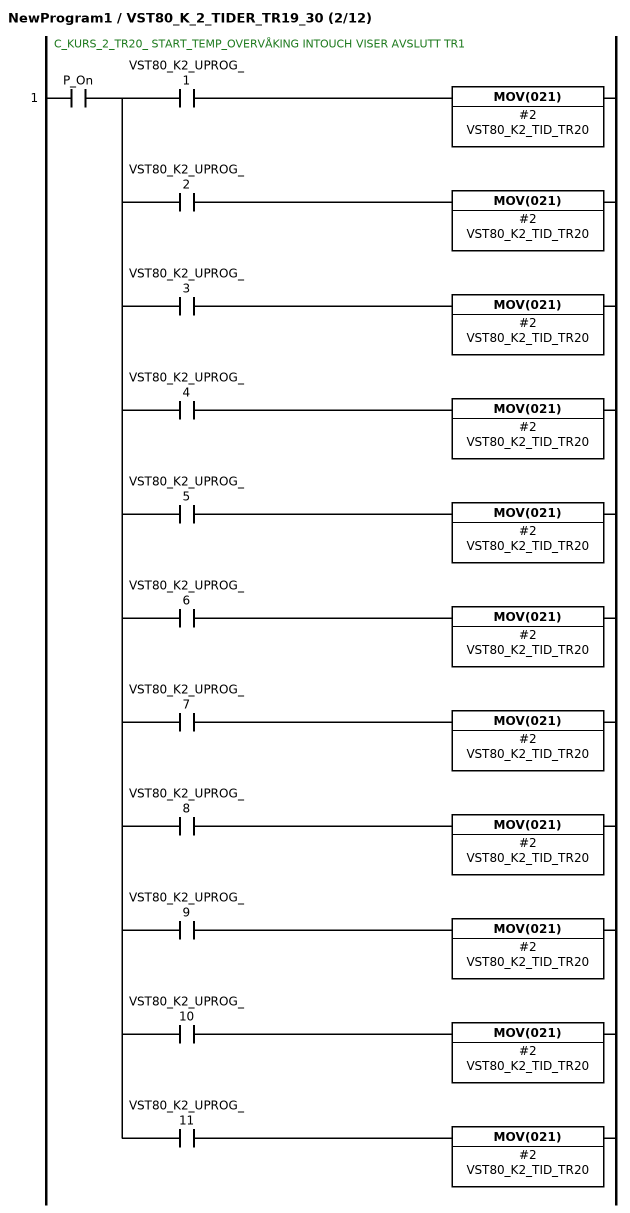
; rung 1: C_KURS_2_TR20_ START_TEMP_OVERVÅKING INTOUCH VISER AVSLUTT TR1
LD P_On
OUT TR0
AND VST80_K2_UPROG_1
MOV(021) #2 VST80_K2_TID_TR20
LD TR0
AND VST80_K2_UPROG_2
MOV(021) #2 VST80_K2_TID_TR20
LD TR0
AND VST80_K2_UPROG_3
MOV(021) #2 VST80_K2_TID_TR20
LD TR0
AND VST80_K2_UPROG_4
MOV(021) #2 VST80_K2_TID_TR20
LD TR0
AND VST80_K2_UPROG_5
MOV(021) #2 VST80_K2_TID_TR20
LD TR0
AND VST80_K2_UPROG_6
MOV(021) #2 VST80_K2_TID_TR20
LD TR0
AND VST80_K2_UPROG_7
MOV(021) #2 VST80_K2_TID_TR20
LD TR0
AND VST80_K2_UPROG_8
MOV(021) #2 VST80_K2_TID_TR20
LD TR0
AND VST80_K2_UPROG_9
MOV(021) #2 VST80_K2_TID_TR20
LD TR0
AND VST80_K2_UPROG_10
MOV(021) #2 VST80_K2_TID_TR20
LD TR0
AND VST80_K2_UPROG_11
MOV(021) #2 VST80_K2_TID_TR20

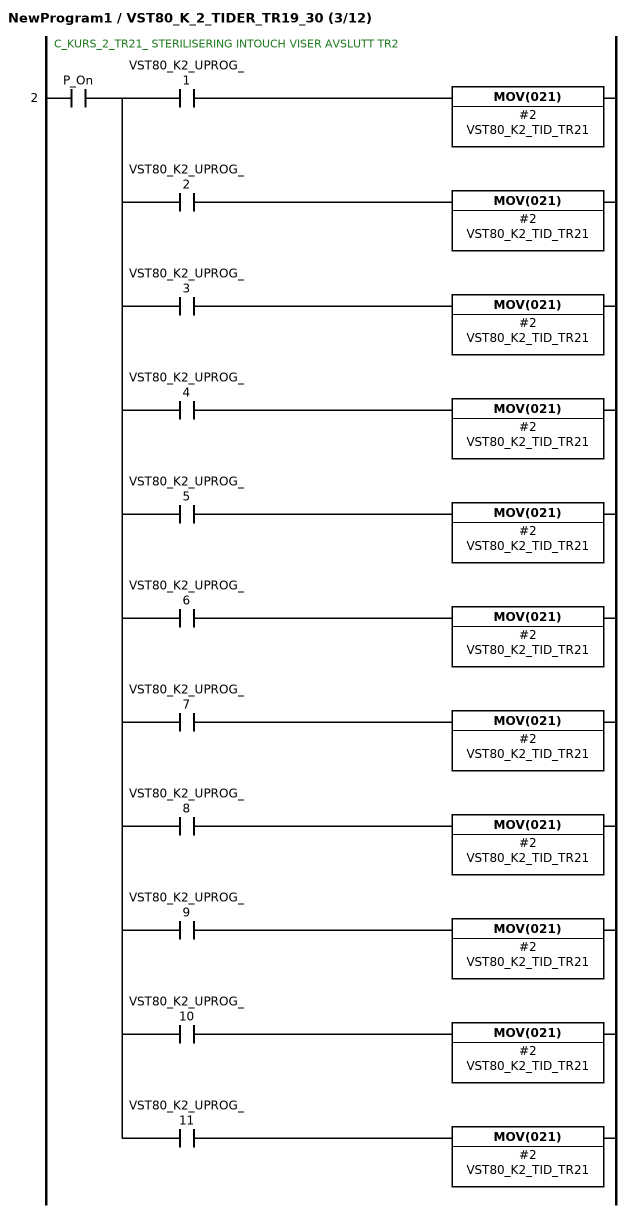
; rung 2: C_KURS_2_TR21_ STERILISERING INTOUCH VISER AVSLUTT TR2
LD P_On
OUT TR0
AND VST80_K2_UPROG_1
MOV(021) #2 VST80_K2_TID_TR21
LD TR0
AND VST80_K2_UPROG_2
MOV(021) #2 VST80_K2_TID_TR21
LD TR0
AND VST80_K2_UPROG_3
MOV(021) #2 VST80_K2_TID_TR21
LD TR0
AND VST80_K2_UPROG_4
MOV(021) #2 VST80_K2_TID_TR21
LD TR0
AND VST80_K2_UPROG_5
MOV(021) #2 VST80_K2_TID_TR21
LD TR0
AND VST80_K2_UPROG_6
MOV(021) #2 VST80_K2_TID_TR21
LD TR0
AND VST80_K2_UPROG_7
MOV(021) #2 VST80_K2_TID_TR21
LD TR0
AND VST80_K2_UPROG_8
MOV(021) #2 VST80_K2_TID_TR21
LD TR0
AND VST80_K2_UPROG_9
MOV(021) #2 VST80_K2_TID_TR21
LD TR0
AND VST80_K2_UPROG_10
MOV(021) #2 VST80_K2_TID_TR21
LD TR0
AND VST80_K2_UPROG_11
MOV(021) #2 VST80_K2_TID_TR21

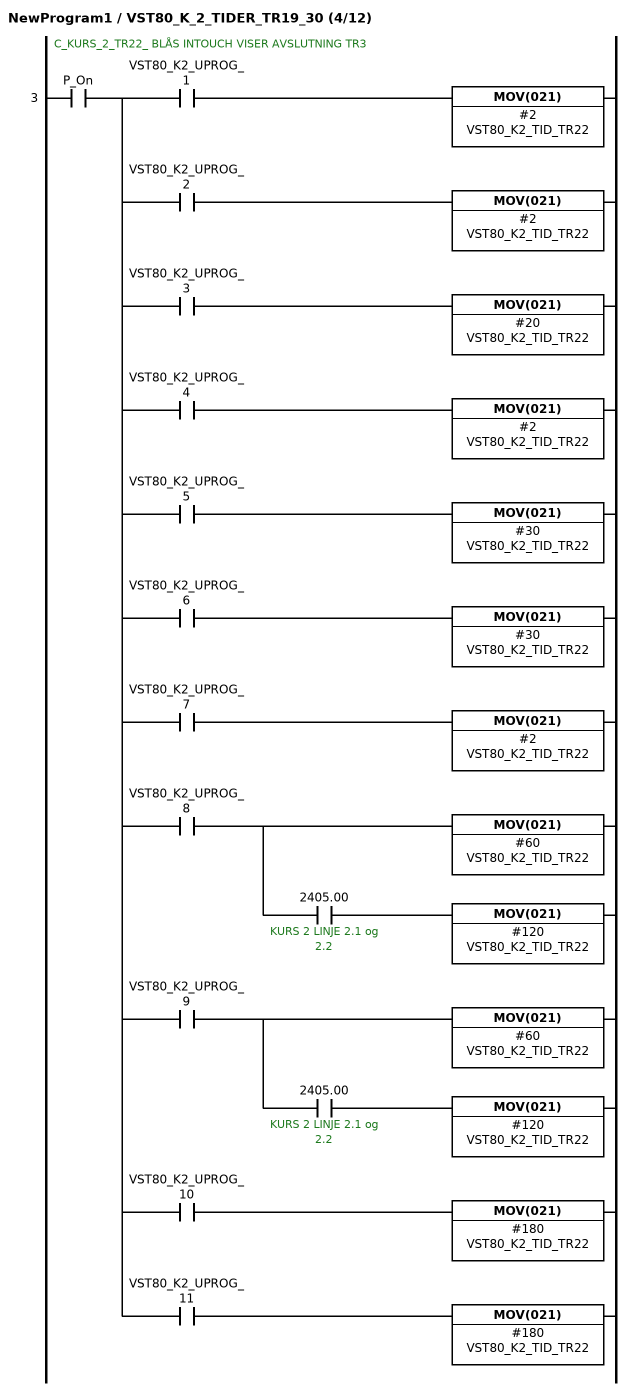
; rung 3: C_KURS_2_TR22_ BLÅS INTOUCH VISER AVSLUTNING TR3
LD P_On
OUT TR0
AND VST80_K2_UPROG_1
MOV(021) #2 VST80_K2_TID_TR22
LD TR0
AND VST80_K2_UPROG_2
MOV(021) #2 VST80_K2_TID_TR22
LD TR0
AND VST80_K2_UPROG_3
MOV(021) #20 VST80_K2_TID_TR22
LD TR0
AND VST80_K2_UPROG_4
MOV(021) #2 VST80_K2_TID_TR22
LD TR0
AND VST80_K2_UPROG_5
MOV(021) #30 VST80_K2_TID_TR22
LD TR0
AND VST80_K2_UPROG_6
MOV(021) #30 VST80_K2_TID_TR22
LD TR0
AND VST80_K2_UPROG_7
MOV(021) #2 VST80_K2_TID_TR22
LD TR0
AND VST80_K2_UPROG_8
MOV(021) #60 VST80_K2_TID_TR22
AND 2405.00  ; KURS 2 LINJE 2.1 og 2.2
MOV(021) #120 VST80_K2_TID_TR22
LD TR0
AND VST80_K2_UPROG_9
MOV(021) #60 VST80_K2_TID_TR22
AND 2405.00  ; KURS 2 LINJE 2.1 og 2.2
MOV(021) #120 VST80_K2_TID_TR22
LD TR0
AND VST80_K2_UPROG_10
MOV(021) #180 VST80_K2_TID_TR22
LD TR0
AND VST80_K2_UPROG_11
MOV(021) #180 VST80_K2_TID_TR22

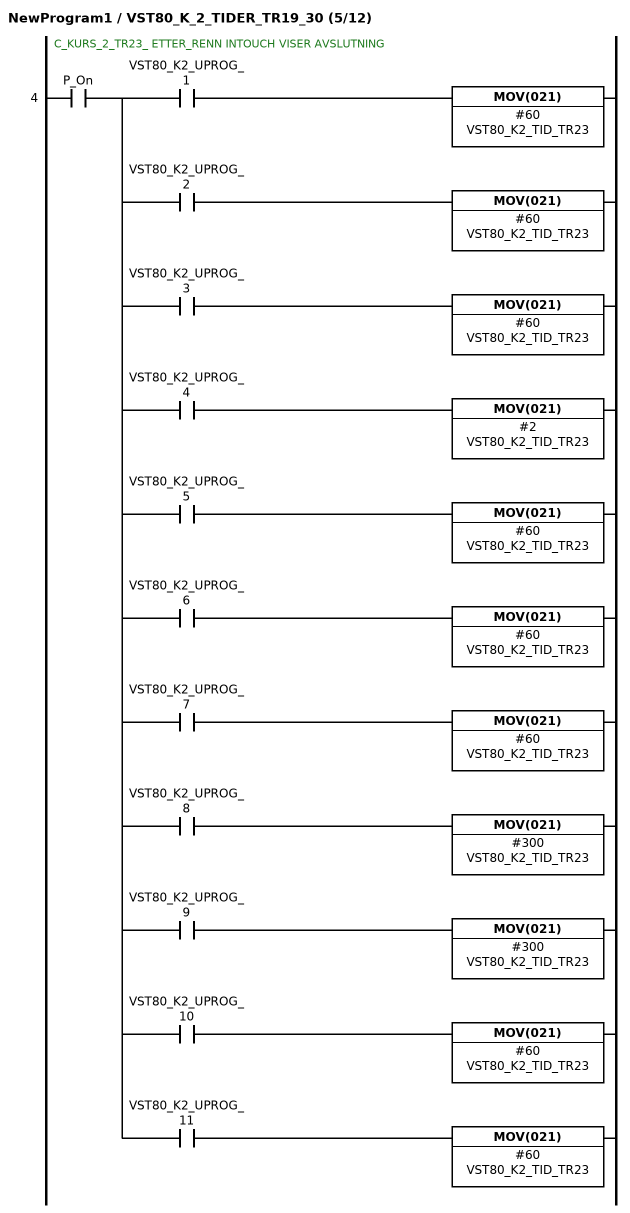
; rung 4: C_KURS_2_TR23_ ETTER_RENN INTOUCH VISER AVSLUTNING
LD P_On
OUT TR0
AND VST80_K2_UPROG_1
MOV(021) #60 VST80_K2_TID_TR23
LD TR0
AND VST80_K2_UPROG_2
MOV(021) #60 VST80_K2_TID_TR23
LD TR0
AND VST80_K2_UPROG_3
MOV(021) #60 VST80_K2_TID_TR23
LD TR0
AND VST80_K2_UPROG_4
MOV(021) #2 VST80_K2_TID_TR23
LD TR0
AND VST80_K2_UPROG_5
MOV(021) #60 VST80_K2_TID_TR23
LD TR0
AND VST80_K2_UPROG_6
MOV(021) #60 VST80_K2_TID_TR23
LD TR0
AND VST80_K2_UPROG_7
MOV(021) #60 VST80_K2_TID_TR23
LD TR0
AND VST80_K2_UPROG_8
MOV(021) #300 VST80_K2_TID_TR23
LD TR0
AND VST80_K2_UPROG_9
MOV(021) #300 VST80_K2_TID_TR23
LD TR0
AND VST80_K2_UPROG_10
MOV(021) #60 VST80_K2_TID_TR23
LD TR0
AND VST80_K2_UPROG_11
MOV(021) #60 VST80_K2_TID_TR23

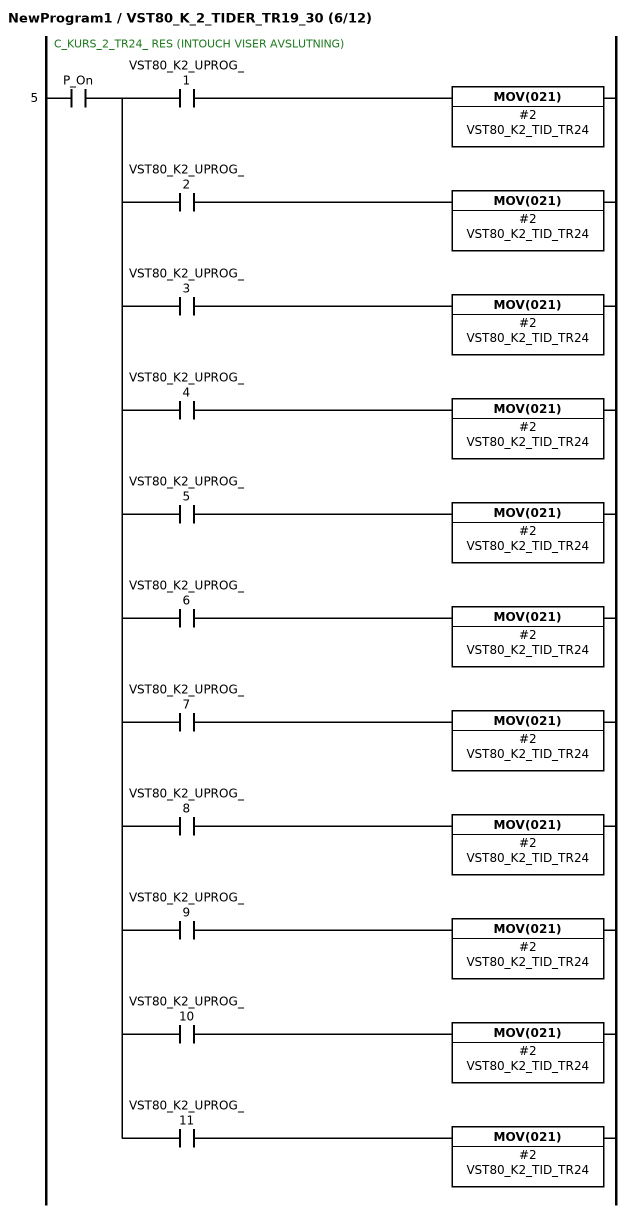
; rung 5: C_KURS_2_TR24_ RES (INTOUCH VISER AVSLUTNING)
LD P_On
OUT TR0
AND VST80_K2_UPROG_1
MOV(021) #2 VST80_K2_TID_TR24
LD TR0
AND VST80_K2_UPROG_2
MOV(021) #2 VST80_K2_TID_TR24
LD TR0
AND VST80_K2_UPROG_3
MOV(021) #2 VST80_K2_TID_TR24
LD TR0
AND VST80_K2_UPROG_4
MOV(021) #2 VST80_K2_TID_TR24
LD TR0
AND VST80_K2_UPROG_5
MOV(021) #2 VST80_K2_TID_TR24
LD TR0
AND VST80_K2_UPROG_6
MOV(021) #2 VST80_K2_TID_TR24
LD TR0
AND VST80_K2_UPROG_7
MOV(021) #2 VST80_K2_TID_TR24
LD TR0
AND VST80_K2_UPROG_8
MOV(021) #2 VST80_K2_TID_TR24
LD TR0
AND VST80_K2_UPROG_9
MOV(021) #2 VST80_K2_TID_TR24
LD TR0
AND VST80_K2_UPROG_10
MOV(021) #2 VST80_K2_TID_TR24
LD TR0
AND VST80_K2_UPROG_11
MOV(021) #2 VST80_K2_TID_TR24

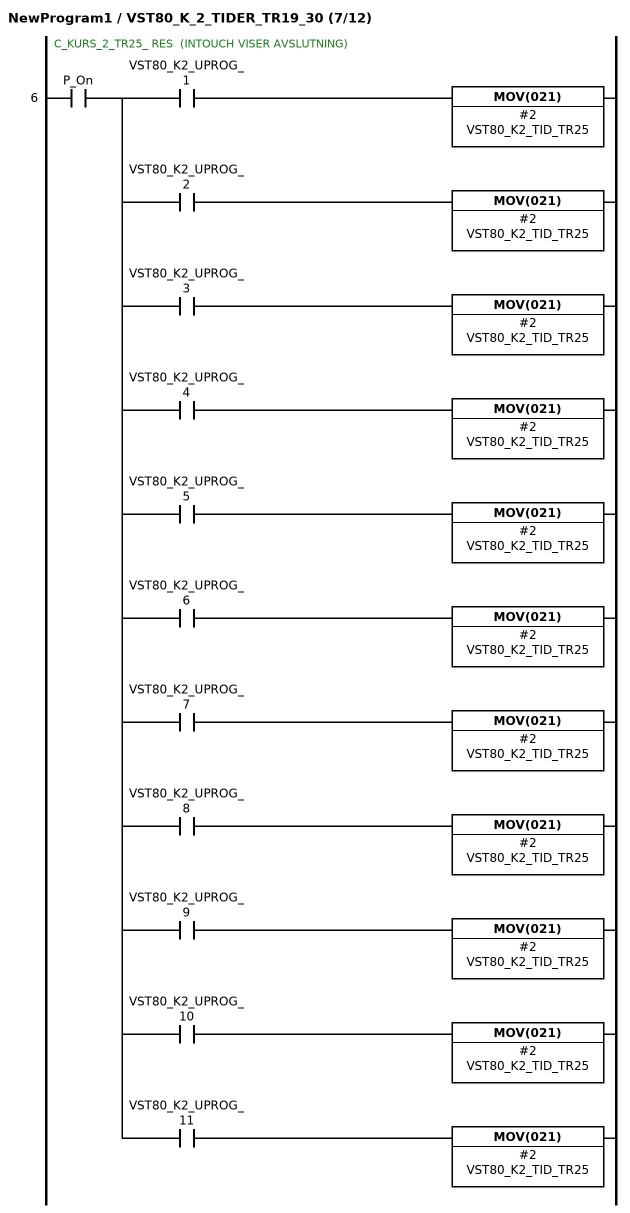
; rung 6: C_KURS_2_TR25_ RES  (INTOUCH VISER AVSLUTNING)
LD P_On
OUT TR0
AND VST80_K2_UPROG_1
MOV(021) #2 VST80_K2_TID_TR25
LD TR0
AND VST80_K2_UPROG_2
MOV(021) #2 VST80_K2_TID_TR25
LD TR0
AND VST80_K2_UPROG_3
MOV(021) #2 VST80_K2_TID_TR25
LD TR0
AND VST80_K2_UPROG_4
MOV(021) #2 VST80_K2_TID_TR25
LD TR0
AND VST80_K2_UPROG_5
MOV(021) #2 VST80_K2_TID_TR25
LD TR0
AND VST80_K2_UPROG_6
MOV(021) #2 VST80_K2_TID_TR25
LD TR0
AND VST80_K2_UPROG_7
MOV(021) #2 VST80_K2_TID_TR25
LD TR0
AND VST80_K2_UPROG_8
MOV(021) #2 VST80_K2_TID_TR25
LD TR0
AND VST80_K2_UPROG_9
MOV(021) #2 VST80_K2_TID_TR25
LD TR0
AND VST80_K2_UPROG_10
MOV(021) #2 VST80_K2_TID_TR25
LD TR0
AND VST80_K2_UPROG_11
MOV(021) #2 VST80_K2_TID_TR25

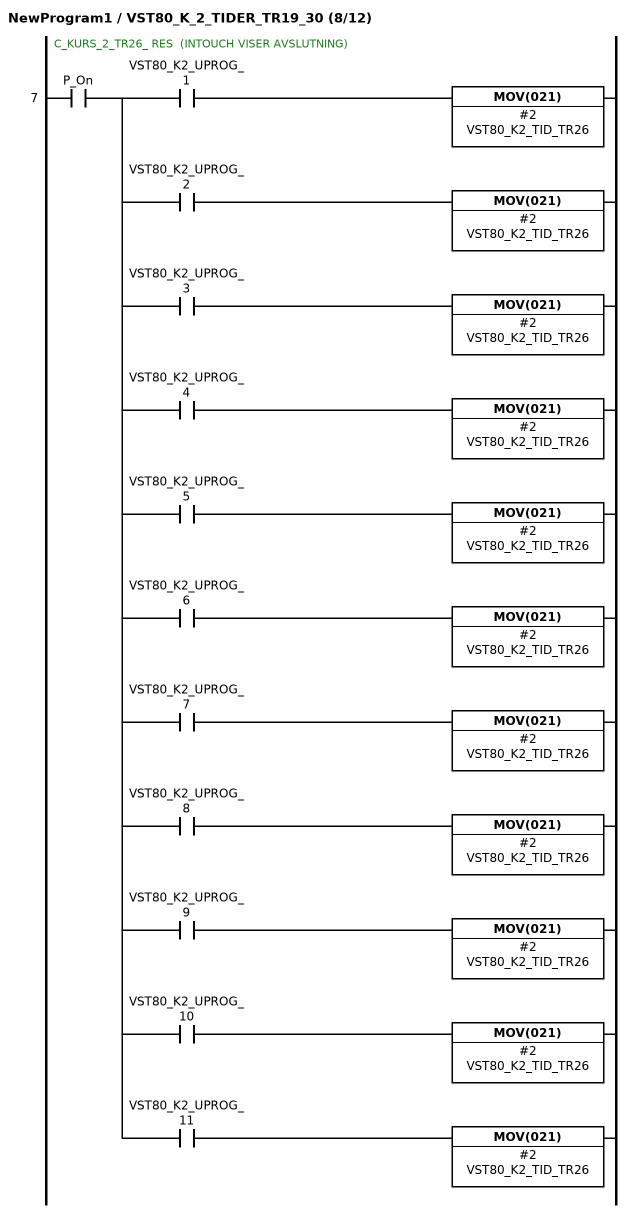
; rung 7: C_KURS_2_TR26_ RES  (INTOUCH VISER AVSLUTNING)
LD P_On
OUT TR0
AND VST80_K2_UPROG_1
MOV(021) #2 VST80_K2_TID_TR26
LD TR0
AND VST80_K2_UPROG_2
MOV(021) #2 VST80_K2_TID_TR26
LD TR0
AND VST80_K2_UPROG_3
MOV(021) #2 VST80_K2_TID_TR26
LD TR0
AND VST80_K2_UPROG_4
MOV(021) #2 VST80_K2_TID_TR26
LD TR0
AND VST80_K2_UPROG_5
MOV(021) #2 VST80_K2_TID_TR26
LD TR0
AND VST80_K2_UPROG_6
MOV(021) #2 VST80_K2_TID_TR26
LD TR0
AND VST80_K2_UPROG_7
MOV(021) #2 VST80_K2_TID_TR26
LD TR0
AND VST80_K2_UPROG_8
MOV(021) #2 VST80_K2_TID_TR26
LD TR0
AND VST80_K2_UPROG_9
MOV(021) #2 VST80_K2_TID_TR26
LD TR0
AND VST80_K2_UPROG_10
MOV(021) #2 VST80_K2_TID_TR26
LD TR0
AND VST80_K2_UPROG_11
MOV(021) #2 VST80_K2_TID_TR26

